# B&R Automation Studio project Lab3_test
Automation Studio 4.5.2.102

## Logical view

Binary libraries used (declarations not repeated): Runtime, Operator, AsIecCon, astime, sys_lib, asstring, Acp10man, Acp10par, NcGlobal, Acp10sdc, Acp10_MC, brsystem, AsBrStr, Acp10sim, AsIOTime

### Global.var - Global variables
```iecst
VAR
	gAxis_X : ACP10AXIS_typ := (0);
	gAxis_X_HW : SdcHwCfg_typ := (0);
	gAxis_X_DrvIf : SdcDrvIf16_typ := (0);
	gAxis_X_DiDoIf : SdcDiDoIf_typ := (0);
	gAxis_X_EncIf : SdcEncIf16_typ := (0);
	gAxis01 : ACP10AXIS_typ := (0);
	gAxis01_HW : SdcHwCfg_typ := (0);
	gAxis01_DrvIf : SdcDrvIf16_typ := (0);
	gAxis01_DiDoIf : SdcDiDoIf_typ := (0);
	gAxis01_ModuleOk : BOOL := 0;
END_VAR
```

### Package Logical/Libraries - Global libraries

### Library Logical/Libraries/MotrContr (ANSIC)

#### MotrContr.fun - Exported functions and function blocks
```iecst
{REDUND_ERROR} {REDUND_UNREPLICABLE} FUNCTION_BLOCK FB_Integrator (*TODO: Add your comment here*) (*$GROUP=User,$CAT=User,$GROUPICON=User.png,$CATICON=User.png*)
	VAR_INPUT
		in : {REDUND_UNREPLICABLE} REAL;
	END_VAR
	VAR_OUTPUT
		out : {REDUND_UNREPLICABLE} REAL;
	END_VAR
	VAR
		dt : {REDUND_UNREPLICABLE} REAL;
	END_VAR
END_FUNCTION_BLOCK

{REDUND_ERROR} {REDUND_UNREPLICABLE} FUNCTION_BLOCK FB_Motor (*TODO: Add your comment here*) (*$GROUP=User,$CAT=User,$GROUPICON=User.png,$CATICON=User.png*)
	VAR_INPUT
		u : {REDUND_UNREPLICABLE} REAL;
	END_VAR
	VAR_OUTPUT
		w : {REDUND_UNREPLICABLE} REAL;
		phi : {REDUND_UNREPLICABLE} REAL;
	END_VAR
	VAR
		integrator : {REDUND_UNREPLICABLE} FB_Integrator;
		Tm : {REDUND_UNREPLICABLE} REAL;
		ke : {REDUND_UNREPLICABLE} REAL;
		dt : {REDUND_UNREPLICABLE} REAL;
	END_VAR
END_FUNCTION_BLOCK

{REDUND_ERROR} FUNCTION_BLOCK FB_Regulator (*TODO: Add your comment here*) (*$GROUP=User,$CAT=User,$GROUPICON=User.png,$CATICON=User.png*)
	VAR_INPUT
		e : {REDUND_UNREPLICABLE} REAL;
	END_VAR
	VAR_OUTPUT
		u : {REDUND_UNREPLICABLE} REAL;
	END_VAR
	VAR
		k_p : {REDUND_UNREPLICABLE} REAL;
		k_i : {REDUND_UNREPLICABLE} REAL;
		integrator : {REDUND_UNREPLICABLE} FB_Integrator;
		iyOld : {REDUND_UNREPLICABLE} REAL;
		max_abs_value : {REDUND_UNREPLICABLE} REAL;
		abs_in_2 : REAL;
		abs_in_1 : REAL;
		abs_out_1 : REAL;
		e_kp : REAL;
		dt : {REDUND_UNREPLICABLE} REAL;
	END_VAR
END_FUNCTION_BLOCK

{REDUND_ERROR} FUNCTION_BLOCK FB_Axis (*TODO: Add your comment here*) (*$GROUP=User,$CAT=User,$GROUPICON=User.png,$CATICON=User.png*)
	VAR_INPUT
		reset_error : BOOL;
		endswitch_a_reached : BOOL;
		endswitch_b_reached : BOOL;
		u : INT;
	END_VAR
	VAR_OUTPUT
		reset_counter : BOOL;
		pwm_value : INT;
		counter : INT;
		speed : REAL;
	END_VAR
	VAR
		last_counter : INT;
	END_VAR
END_FUNCTION_BLOCK
```

#### FB_Motor.c
```c
#include <bur/plctypes.h>
#ifdef __cplusplus
	extern "C"
	{
#endif
	#include "MotrContr.h"
#ifdef __cplusplus
	};
#endif
/* TODO: Add your comment here */
void FB_Motor(struct FB_Motor* inst)
{
	inst->integrator.in = (inst->u / inst->ke - inst->w) * inst->dt / inst->Tm; //integr's in (incoming signal u multipled by 1/ke subtracting w then multipled by dt/Tm)

	//inst->integrator.out = inst->w;

	FB_Integrator(&(inst->integrator));			//calling integr
	inst->w = inst->integrator.out;				//from 1 integr

	inst->integrator.in = inst->w * inst->dt;	//integr's in (incoming signal w multipled by dt)

	//inst->integrator.out = inst->phi;

	FB_Integrator(&(inst->integrator));			//calling integr

	inst->phi = inst->integrator.out; 			//outcoming signal phi
}
```

#### FB_Regulator.c
```c
#include <bur/plctypes.h>
#ifdef __cplusplus
	extern "C"
	{
#endif
	#include "MotrContr.h"
#ifdef __cplusplus
	};
#endif
/* TODO: Add your comment here */
void FB_Regulator(struct FB_Regulator* inst)
{

	/*
	inst->integrator.in = inst->e * inst->k_i * inst->dt + inst->iyOld;	//integr's in (incoming signal e multipled by ki and dt adding old value)
	FB_Integrator(&(inst->integrator));			//calling integr

	inst->abs_in_1 = inst->e * inst->k_p;		//limiter's in

	if(inst->abs_in_1 > inst->max_abs_value || inst->abs_in_1 < -inst->max_abs_value)	//if in is equal or more than limit
		{
			if(inst->abs_in_1 > 0)
			{
				inst->abs_out_1 = inst->max_abs_value;	//than limit the value
			}
			else
			{
				inst->abs_out_1 = -inst->max_abs_value;	//than limit the value
			}
	}
	else 										//else if in is less than limit
	{
		inst->abs_out_1 = inst->abs_in_1;		//than transmit the value to limiter's out
	}

	inst->abs_in_2 = inst->abs_out_1 + inst->integrator.out;	//transmit summ of integral and proport parts to limiter's in

	if(inst->abs_in_2 > inst->max_abs_value || inst->abs_in_2 < -inst->max_abs_value)		//if in is equal or more than limit
	{
		if(inst->abs_in_2 > 0)
		{
			inst->u = inst->max_abs_value;			//than limit the value and set to the outcoming signal u
		}
		else
		{
			inst->u = -inst->max_abs_value;			//than limit the value and set to the outcoming signal u
		}
	}
	else 										//else if in is less than limit
	{
		inst->u = inst->abs_in_2;				//than transmit the value to limiter's out and set to the outcoming signal u
	}

	inst->iyOld = inst->u - inst->abs_in_2;		//saving the current value

	*/

	inst->integrator.in=inst->e * inst->k_i * inst->dt + inst->iyOld;

	FB_Integrator(&(inst->integrator));

	inst->e_kp=inst->e*inst->k_p;

	inst->e_kp=(inst->e_kp > inst->max_abs_value || inst->e_kp < - inst->max_abs_value)?((inst->e_kp>0)?inst->max_abs_value:-inst->max_abs_value):inst->e_kp;

	inst->e_kp+=inst->integrator.out;

	inst->u=(inst->e_kp > inst->max_abs_value || inst->e_kp < - inst->max_abs_value)?((inst->e_kp>0)?inst->max_abs_value:-inst->max_abs_value):inst->e_kp;

	inst->iyOld=inst->u-inst->e_kp;

}
```

#### FB_Integrator.c
```c
#include <bur/plctypes.h>
#ifdef __cplusplus
	extern "C"
	{
#endif
	#include "MotrContr.h"
#ifdef __cplusplus
	};
#endif
/* TODO: Add your comment here */
void FB_Integrator(struct FB_Integrator* inst)
{
	inst->out += inst->in /* inst->dt*/;
}
```

#### FB_Axis.c
```c
#include <bur/plctypes.h>
#ifdef __cplusplus
	extern "C"
	{
#endif
	#include "MotrContr.h"
#ifdef __cplusplus
	};
#endif
/* TODO: Add your comment here */
void FB_Axis(struct FB_Axis* inst)
{
	if (inst->endswitch_a_reached || inst->endswitch_b_reached)
	{
		inst->pwm_value=0;
		inst->reset_error=1;
	}
	else
	{
		inst->pwm_value=inst->u/24.0*32767;//шим соответственно напряжению с регулятора
		inst->reset_error=0;
	}
	inst->speed=inst->u/24.0*6500.0;
}
```

Listed in the project but not available here: Logical/Global.typ, Logical/Libraries/MotrContr/Types.typ, Logical/Libraries/MotrContr/Constants.var, Logical/acp10etxen, Logical/SDCAxisCtrlX, Logical/ncsdcctrl, Logical/gAxis01obj
